// TIA Portal V19 export
TYPE "LEXCHANGETRAY_typeRollerIoSignalControlNode"
// reset: Bool
// monitoring: LEXCHANGETRAY_typeRollerIoSignalContronNodeMonitoring
// stored: Access Published
   STRUCT
      reset : Bool;
      monitoring { S7_SetPoint := 'True'} : "LEXCHANGETRAY_typeRollerIoSignalContronNodeMonitoring";
   END_STRUCT;
END_TYPE
